TYPE STATE:
    STRUCT
        curTime: REAL;
        cvar_c: REAL;
        dvar_M_aut_r: REAL;
        dvar_M_aut_b: BOOL;
        dvar_M_aut_i: DINT;
        dvar_M_aut_tii: TupleStruct_1;
        dvar_M_aut_i2: DINT;
        dvar_M_aut_i3: DINT;
        dvar_M_aut: DINT;
    END_STRUCT;
END_TYPE
